{attribute addProperty BoxType "EL6001--0000"}
{attribute addProperty Id "StatusAT %I*UINT1621Data_InAT %I*ARRAY[0 ..21] OF USINT176220"}
{attribute addProperty CRC "2032034109"}
{attribute addProperty SizeInBites "192"}
{attribute addProperty SizeInBytes "24"}
TYPE Inputs_DD54DA92 :
STRUCT
	{attribute addProperty Name "Status"}
	Status AT %I* : UINT;
	{attribute addProperty Name "Data_In"}
	Data_In AT %I* : ARRAY[0 ..21] OF USINT;
END_STRUCT
END_TYPE

(* stored: Version 1.2.0.0, ProductVersion 3.1.4024.9
   DUT Inputs_DD54DA92: Id {0a2abfab-7de5-40ca-9e11-b20b04c591f6} *)
